// TIA Portal project "Ejemplo_III" (V16)

(* hardware
DEVICE "PC-System_1"  SIMATIC PC station
   slot 0: "Estación PC SIMATIC"  Rail  SIMATIC PC-Station  V1.0
      slot 125: "Stationmanager"  Station_Manager  V6.0.4
   slot 1: "HMI_RT_1"  WinCC RT Advanced  6AV2 104-0xxxx-xxxx  16.0.0.0
      slot 33792: "Interfaz del equipo"  Host interface
   slot 2: "IE general_1"  IE General  IE_CP  V8.2.0
DEVICE "S7300/ET200M station_1"  S7-300 station
   slot 0: "Perfil soporte_0"  Rail  6ES7 390-1***0-0AA0
   slot 2: "PLC_1"  CPU 313C  6ES7 313-5BG04-0AB0  V3.3
      slot 0: "Interfaz MPI_1"  MPI
      slot 2: "DI 24/DO 16_1"  DI24/DO16
      slot 3: "AI 5/AO 2_1"  AI5/AO2
      slot 4: "Contaje_1"  Counter
   slot 4: "CP 343-1 Lean_1"  CP 343-1 LEAN  6GK7 343-1CX10-0XE0  V3.0
*)

// ===== PLC "PLC_1"  CPU 313C =====

DATA_BLOCK "Bloque de datos_1"   // DB1
{ S7_Optimized_Access := 'FALSE' }
VERSION : 0.1
   VAR
      Memoria : Bool;
      Memoria_real : Real;
      Memoria_entera : Int;
   END_VAR
BEGIN
END_DATA_BLOCK

ORGANIZATION_BLOCK "Main"   // OB1, LAD
TITLE = "Main Program Sweep (Cycle)"
{ S7_Optimized_Access := 'FALSE' }
VERSION : 0.1
   VAR_TEMP
      OB1_EV_CLASS : Byte;   // Bits 0-3 = 1 (Coming event), Bits 4-7 = 1 (Event class 1)
      OB1_SCAN_1 : Byte;   // 1 (Cold restart scan 1 of OB 1), 3 (Scan 2-n of OB 1)
      OB1_PRIORITY : Byte;   // Priority of OB Execution
      OB1_OB_NUMBR : Byte;   // 1 (Organization block 1, OB1)
      OB1_RESERVED_1 : Byte;   // Reserved for system
      OB1_RESERVED_2 : Byte;   // Reserved for system
      OB1_PREV_CYCLE : Int;   // Cycle time of previous OB1 scan (milliseconds)
      OB1_MIN_CYCLE : Int;   // Minimum cycle time of OB1 (milliseconds)
      OB1_MAX_CYCLE : Int;   // Maximum cycle time of OB1 (milliseconds)
      OB1_DATE_TIME : Date_And_Time;   // Date and time OB1 started
   END_VAR
BEGIN
END_ORGANIZATION_BLOCK

(* ===== HMI "HMI_RT_1" =====
system functions are stored by id; their names below are inferred from use
connection "HMI_Conexión_1": ETHERNET, SIMATIC S7 300/400 MPI

HMI tags "Tabla de variables estándar"
   "Variable_Booleana" : Bool = PLC "Bloque de datos_1".Memoria AT %DB1.DBX0.0, 1 s
   "Variable_Real" : Real = PLC "Bloque de datos_1".Memoria_real AT %DB1.DBD2, 1 s
   "Variable_Entera" : Int = PLC "Bloque de datos_1".Memoria_entera AT %DB1.DBW6, 1 s
   "Variable_prueba" : Real, internal

screen "Imagen_1" 800x600
   Button "Botón_1" at 285,332 size 96x32; TextOff 'Boton1'
      on Press: "Acumulador"()
   Button "Botón_2" at 285,408 size 96x32; TextOff 'Boton2'
      on Press: "Exportar"()
   IOField "Campo ES_1" at 419,332 size 96x32; FormatPattern s999999999.999
      ProcessValue <- "Variable_prueba"

VB script "Basico"
   'Variables Globales
   SmartTags("Variable_prueba") = 0
   'Variables en VB (locales)
   Dim Variable1, Variable2, Variable3, Variablen
   Variable1 = 5 'Entera
   Variable2 = 12.4 'Decimal
   Variable3 = #12:30:22 PM# 'Hora
   Variablen = "Hola mundo"
   'Arreglo
   Dim Vector
   Vector = Array(1, 2, 3)
   'Operaciones matemàticas
   Dim Res
   Res = Variable1+Variable2
   Res = Variable1-Variable2
   Res = Variable1*Variable2
   Res = Variable1/Variable2
   
   SmartTags("Variable_prueba") = Res

VB script "Boton1"
   SmartTags("Variable_Booleana") = False
   SmartTags("Variable_Real") = 10
   SmartTags("Variable_Entera") = 300

VB script "Boton2"
   SmartTags("Variable_Booleana") = True
   SmartTags("Variable_Real") = 15.5
   SmartTags("Variable_Entera") = 44

VB script "Acumulador"
   'Sugerencia:
   ' 1. Utilice la combinación de teclas <CTRL+ESPACIO> o <CTRL+I> para abrir una lista de todos los objetos y funciones
   ' 2. Escriba el código utilizando el objeto HMI Runtime.
   '  Ejemplo: HmiRuntime.Screens("Screen_1").
   ' 3. Utilice la combinación de teclas <CTRL+J> para crear una referencia de objeto..
   'Escriba el código a partir de esta posición:
   Dim Aux
   Aux=5
   SmartTags("Variable_prueba")=SmartTags("Variable_prueba")+Aux

VB script "Control_Flujo"
   'Condicional if-else
   Dim condicion
   condicion = 10
   If condicion = 10 Then
   	SmartTags("Variable_prueba")=1
   Else
   	SmartTags("Variable_prueba")=0
   End If
   '=  Comparacion
   '<> Distinto de
   '>= Mayor o igual
   '<= Menor o igual
   'Iterativas 
   Do Until condicion = 0 'Do Until (Haga hasta que...)
   	condicion = condicion-1
   Loop
   'Dim contador
   'For contador = 0 To 5 Step 1 'For
   '	SmartTags("Variable_prueba")=contador
   'Next
   
   'Ej2. Llenado de un Vector
   Dim contador
   Dim Vector(5)
   For contador = 0 To 5 Step 1 
   	Vector(contador)=contador
   Next
   'Ej3. Llenado de una Matriz
   Dim i, j
   Dim Matriz(3,3)
   For i = 0 To 3 Step 1 
   	For j = 0 To 3 Step 1 
   		Matriz(i,j)=j
   	Next
   Next
   'Ej4. Delay
   Dim Futuro
   Dim Espera
   Espera = 10 'Segundos
   Futuro = DateAdd("s", Espera, Now())
   Do Until(Now()>Futuro)
   Loop

VB script "Exportar"
   Dim Ruta, Objeto, Objeto2
   Ruta = "C:/Archivo.csv"
   'Objeto para el archivo
   Set Objeto = CreateObject("Scripting.FileSystemObject")
   '1-Leer, 2-Escribir, 8-Agregar
   Set Objeto2 = Objeto.OpenTextFile(Ruta, 8, True)
   'Concatenar cadena de salida
   Dim dato
   dato=Now & ";" & SmartTags("Variable_prueba")
   Objeto2.WriteLine dato
   Objeto2.Close
   Set Objeto = Nothing
   Set Objeto2 = Nothing
*)